INTERFACE Proxy_Interface

///Illustrative method of the pattern
METHOD Set_Background
VAR_INPUT
	///HEX value to be set as background color
	newBackground: DWORD;
END_VAR
END_METHOD

END_INTERFACE

(* stored: Version 1.1.0.1, ProductVersion 3.1.4024.11
   Itf Proxy_Interface: Id {c09f41ed-8388-4fa5-846b-482111779151}
   Method Set_Background: Id {0b61ddc6-a83a-488f-9e3c-0f6b2e254ece} *)
